//INTERFACE ITcoDriveSimple EXTENDS TcoCore.ITcoComponent
INTERFACE ITcoDriveSimple

PROPERTY DriveRef : REFERENCE TO TcoDriveSimple
GET
END_GET
END_PROPERTY

END_INTERFACE

(* stored: Version 1.1.0.1, ProductVersion 3.1.4024.6
   Itf ITcoDriveSimple: Id {6fdf7305-86e5-0f64-03c7-4bbd6de45ddc}
   Property DriveRef: Id {cf2de1bd-d6db-0dcf-3c72-d4602879a41f}
   Get Get: Id {275430ab-40ad-0ea1-0981-550561d9b0a4} *)
